FUNCTION_BLOCK FB_Beckhoff_EL5152_Test EXTENDS TcUnit.FB_TestSuite
VAR
	_fbDevice 	: FB_Beckhoff_EL5152;
	_nExpected 	: UINT;
	_nResult 	: UINT;
END_VAR

TEST('nCounter1');
_nExpected := 111;
_fbDevice.nValue1 := _nExpected;
_fbDevice();
_nResult := _fbDevice.Counter1;
AssertEquals(Expected := _nExpected,
             Actual := _nResult,
             Message := 'nCounter1 value is not correct');	
TEST_FINISHED();

TEST('nCounter2');
_nExpected := 112;
_fbDevice.nValue2 := _nExpected;
_fbDevice();
_nResult := _fbDevice.Counter2;
AssertEquals(Expected := _nExpected,
             Actual := _nResult,
             Message := 'nCounter2 value is not correct');	
TEST_FINISHED();


TEST('nStatus1');
_nExpected := 4;
_fbDevice.Control1 := _nExpected;
_fbDevice();
_nResult := _fbDevice.Status1;
AssertEquals(Expected := _nExpected,
             Actual := _nResult,
             Message := 'nStatus1 value is not correct');	
TEST_FINISHED();

TEST('nStatus2');
_nExpected := 4;
_fbDevice.Control2 := _nExpected;
_fbDevice();
_nResult := _fbDevice.Status2;
AssertEquals(Expected := _nExpected,
             Actual := _nResult,
             Message := 'nStatus2 value is not correct');	
TEST_FINISHED();

END_FUNCTION_BLOCK

(* stored: Version 1.1.0.1, ProductVersion 3.1.4024.12
   POU FB_Beckhoff_EL5152_Test: Id {41eadc21-428a-091f-0416-55b3c1826864}, SpecialFunc None *)
